KUKA KRL data list: hp251.dat

&ACCESS RVP
&REL 2
&COMMENT Teste de Masterizacao
&PARAM TEMPLATE = C:\KRC\ROBOTER\TEMPLATE\VG_HP
&PARAM EDITMASK = *
DEFDAT hp251
;FOLD EXTERNAL DECLARATIONS;%{PE}%MKUKATPBASIS,%CEXT,%VCOMMON,%P
   ;FOLD GRIPPERTECH EXT
      EXT  H50 (INT  :IN,INT  :IN,INT  :IN,GRP_TYP  :IN )
   ;ENDFOLD (GRIPPERTECH EXT)
   ;FOLD SPOTTECH EXT
      EXT  USERSPOT (S_COMMAND  :IN,SPOT_TYPE  :IN )
   ;ENDFOLD (SPOTTECH EXT)
   ;FOLD BASISTECH EXT;%{PE}%MKUKATPBASIS,%CEXT,%VEXT,%P
      EXT  BAS (BAS_COMMAND  :IN,REAL  :IN )
      DECL INT SUCCESS
   ;ENDFOLD (BASISTECH EXT)
   ;FOLD USER EXT;%{E}%MKUKATPUSER,%CEXT,%VEXT,%P
      ;Make your modifications here

   ;ENDFOLD (USER EXT)
;ENDFOLD (EXTERNAL DECLARATIONS)

ENDDAT
